// TIA Portal V17 export
// export: Created 2025-03-07T09:19:28.6491986Z, ExportSetting WithDefaults, DisplayName Totally Integrated Automation Portal, DisplayVersion V17 Update 8, DisplayName TIA Portal Openness, DisplayVersion V17 Update 8, DisplayName TIA Portal Version Control Interface, DisplayVersion V17, DisplayName SINAMICS Startdrive Advanced, DisplayVersion V17 SP2, DisplayName SINAMICS Startdrive G110M, G120, G120C, G120D, G120P, G115D, DisplayVersion V17 SP2, DisplayName SINAMICS Startdrive G130, G150, S120, S150, SINAMICS MV, S210, DisplayVersion V17 SP2, DisplayName STEP 7 Professional, DisplayVersion V17 Update 8, DisplayName SINUMERIK ONE STEP 7 Toolbox, DisplayVersion V17 Update 12, DisplayName SINUMERIK 840D sl STEP 7 Toolbox, DisplayVersion V17 Update 12, DisplayName STEP 7 Safety, DisplayVersion V17 Update 6, DisplayName WinCC Advanced, DisplayVersion V17 Update 8
TYPE "LBP_typeTMMagazines"
TITLE = Tool management magazines / Almacenes de gestión de herramientas / Magazine zur Werkzeugverwaltung
// User data type to store the magazine data / Tipo de datos de usuario para guardar los datos de almacén / Anwender-Datentyp zum Speichern der Magazindaten
// stored: IsFailsafeCompliant false
   STRUCT
      MaxSpindleNumber : UInt;   // Maximale Spindelanzahl / Maximum spindle number / Número máximo de cabezales
      NumberOfMagazines : UInt;   // Anzahl aller Magazine einschließlich Belade- und Zwischenspeichermagazine / Number of all magazines including loading and buffer magazines / Número total de almacenes, incluidos almacenes de carga e intermedios
      Magazines : Array[1..64] of Struct   // Alle Magazine einschließlich Belade- und Zwischenspeichermagazine / All magazines including loading and buffer magazines / Todos los almacenes, incluidos almacenes de carga e intermedios
         Number : UInt;   // Magazin-Nummer / Magazine number / Número de almacén
         "Type" : UInt;   // Magazintyp / Magazine type / Tipo de almacén
         Places : UInt;   // Anzahl der Plätze im Magazin / Number of locations in magazine / Número de puestos en el almacén
         TMNumber : UInt;   // Werkzeug-Verwaltungsnummer / Tool management number / Número de gestión de herramientas
      END_STRUCT;
   END_STRUCT;
   // // Magazines[2].Number : Magazin-Nummer / Magazine number / Número de almacén
   // // Magazines[3].Number : Magazin-Nummer / Magazine number / Número de almacén
   // // Magazines[4].Number : Magazin-Nummer / Magazine number / Número de almacén
   // // Magazines[5].Number : Magazin-Nummer / Magazine number / Número de almacén
   // // Magazines[6].Number : Magazin-Nummer / Magazine number / Número de almacén
   // // Magazines[7].Number : Magazin-Nummer / Magazine number / Número de almacén
   // // Magazines[8].Number : Magazin-Nummer / Magazine number / Número de almacén
   // // Magazines[9].Number : Magazin-Nummer / Magazine number / Número de almacén
   // // Magazines[10].Number : Magazin-Nummer / Magazine number / Número de almacén
   // // Magazines[11].Number : Magazin-Nummer / Magazine number / Número de almacén
   // // Magazines[12].Number : Magazin-Nummer / Magazine number / Número de almacén
   // // Magazines[13].Number : Magazin-Nummer / Magazine number / Número de almacén
   // // Magazines[14].Number : Magazin-Nummer / Magazine number / Número de almacén
   // // Magazines[15].Number : Magazin-Nummer / Magazine number / Número de almacén
   // // Magazines[16].Number : Magazin-Nummer / Magazine number / Número de almacén
   // // Magazines[17].Number : Magazin-Nummer / Magazine number / Número de almacén
   // // Magazines[18].Number : Magazin-Nummer / Magazine number / Número de almacén
   // // Magazines[19].Number : Magazin-Nummer / Magazine number / Número de almacén
   // // Magazines[20].Number : Magazin-Nummer / Magazine number / Número de almacén
   // // Magazines[21].Number : Magazin-Nummer / Magazine number / Número de almacén
   // // Magazines[22].Number : Magazin-Nummer / Magazine number / Número de almacén
   // // Magazines[23].Number : Magazin-Nummer / Magazine number / Número de almacén
   // // Magazines[24].Number : Magazin-Nummer / Magazine number / Número de almacén
   // // Magazines[25].Number : Magazin-Nummer / Magazine number / Número de almacén
   // // Magazines[26].Number : Magazin-Nummer / Magazine number / Número de almacén
   // // Magazines[27].Number : Magazin-Nummer / Magazine number / Número de almacén
   // // Magazines[28].Number : Magazin-Nummer / Magazine number / Número de almacén
   // // Magazines[29].Number : Magazin-Nummer / Magazine number / Número de almacén
   // // Magazines[30].Number : Magazin-Nummer / Magazine number / Número de almacén
   // // Magazines[31].Number : Magazin-Nummer / Magazine number / Número de almacén
   // // Magazines[32].Number : Magazin-Nummer / Magazine number / Número de almacén
   // // Magazines[33].Number : Magazin-Nummer / Magazine number / Número de almacén
   // // Magazines[34].Number : Magazin-Nummer / Magazine number / Número de almacén
   // // Magazines[35].Number : Magazin-Nummer / Magazine number / Número de almacén
   // // Magazines[36].Number : Magazin-Nummer / Magazine number / Número de almacén
   // // Magazines[37].Number : Magazin-Nummer / Magazine number / Número de almacén
   // // Magazines[38].Number : Magazin-Nummer / Magazine number / Número de almacén
   // // Magazines[39].Number : Magazin-Nummer / Magazine number / Número de almacén
   // // Magazines[40].Number : Magazin-Nummer / Magazine number / Número de almacén
   // // Magazines[41].Number : Magazin-Nummer / Magazine number / Número de almacén
   // // Magazines[42].Number : Magazin-Nummer / Magazine number / Número de almacén
   // // Magazines[43].Number : Magazin-Nummer / Magazine number / Número de almacén
   // // Magazines[44].Number : Magazin-Nummer / Magazine number / Número de almacén
   // // Magazines[45].Number : Magazin-Nummer / Magazine number / Número de almacén
   // // Magazines[46].Number : Magazin-Nummer / Magazine number / Número de almacén
   // // Magazines[47].Number : Magazin-Nummer / Magazine number / Número de almacén
   // // Magazines[48].Number : Magazin-Nummer / Magazine number / Número de almacén
   // // Magazines[49].Number : Magazin-Nummer / Magazine number / Número de almacén
   // // Magazines[50].Number : Magazin-Nummer / Magazine number / Número de almacén
   // // Magazines[51].Number : Magazin-Nummer / Magazine number / Número de almacén
   // // Magazines[52].Number : Magazin-Nummer / Magazine number / Número de almacén
   // // Magazines[53].Number : Magazin-Nummer / Magazine number / Número de almacén
   // // Magazines[54].Number : Magazin-Nummer / Magazine number / Número de almacén
   // // Magazines[55].Number : Magazin-Nummer / Magazine number / Número de almacén
   // // Magazines[56].Number : Magazin-Nummer / Magazine number / Número de almacén
   // // Magazines[57].Number : Magazin-Nummer / Magazine number / Número de almacén
   // // Magazines[58].Number : Magazin-Nummer / Magazine number / Número de almacén
   // // Magazines[59].Number : Magazin-Nummer / Magazine number / Número de almacén
   // // Magazines[60].Number : Magazin-Nummer / Magazine number / Número de almacén
   // // Magazines[61].Number : Magazin-Nummer / Magazine number / Número de almacén
   // // Magazines[62].Number : Magazin-Nummer / Magazine number / Número de almacén
   // // Magazines[63].Number : Magazin-Nummer / Magazine number / Número de almacén
   // // Magazines[64].Number : Magazin-Nummer / Magazine number / Número de almacén
   // // Magazines[2]."Type" : Magazintyp / Magazine type / Tipo de almacén
   // // Magazines[3]."Type" : Magazintyp / Magazine type / Tipo de almacén
   // // Magazines[4]."Type" : Magazintyp / Magazine type / Tipo de almacén
   // // Magazines[5]."Type" : Magazintyp / Magazine type / Tipo de almacén
   // // Magazines[6]."Type" : Magazintyp / Magazine type / Tipo de almacén
   // // Magazines[7]."Type" : Magazintyp / Magazine type / Tipo de almacén
   // // Magazines[8]."Type" : Magazintyp / Magazine type / Tipo de almacén
   // // Magazines[9]."Type" : Magazintyp / Magazine type / Tipo de almacén
   // // Magazines[10]."Type" : Magazintyp / Magazine type / Tipo de almacén
   // // Magazines[11]."Type" : Magazintyp / Magazine type / Tipo de almacén
   // // Magazines[12]."Type" : Magazintyp / Magazine type / Tipo de almacén
   // // Magazines[13]."Type" : Magazintyp / Magazine type / Tipo de almacén
   // // Magazines[14]."Type" : Magazintyp / Magazine type / Tipo de almacén
   // // Magazines[15]."Type" : Magazintyp / Magazine type / Tipo de almacén
   // // Magazines[16]."Type" : Magazintyp / Magazine type / Tipo de almacén
   // // Magazines[17]."Type" : Magazintyp / Magazine type / Tipo de almacén
   // // Magazines[18]."Type" : Magazintyp / Magazine type / Tipo de almacén
   // // Magazines[19]."Type" : Magazintyp / Magazine type / Tipo de almacén
   // // Magazines[20]."Type" : Magazintyp / Magazine type / Tipo de almacén
   // // Magazines[21]."Type" : Magazintyp / Magazine type / Tipo de almacén
   // // Magazines[22]."Type" : Magazintyp / Magazine type / Tipo de almacén
   // // Magazines[23]."Type" : Magazintyp / Magazine type / Tipo de almacén
   // // Magazines[24]."Type" : Magazintyp / Magazine type / Tipo de almacén
   // // Magazines[25]."Type" : Magazintyp / Magazine type / Tipo de almacén
   // // Magazines[26]."Type" : Magazintyp / Magazine type / Tipo de almacén
   // // Magazines[27]."Type" : Magazintyp / Magazine type / Tipo de almacén
   // // Magazines[28]."Type" : Magazintyp / Magazine type / Tipo de almacén
   // // Magazines[29]."Type" : Magazintyp / Magazine type / Tipo de almacén
   // // Magazines[30]."Type" : Magazintyp / Magazine type / Tipo de almacén
   // // Magazines[31]."Type" : Magazintyp / Magazine type / Tipo de almacén
   // // Magazines[32]."Type" : Magazintyp / Magazine type / Tipo de almacén
   // // Magazines[33]."Type" : Magazintyp / Magazine type / Tipo de almacén
   // // Magazines[34]."Type" : Magazintyp / Magazine type / Tipo de almacén
   // // Magazines[35]."Type" : Magazintyp / Magazine type / Tipo de almacén
   // // Magazines[36]."Type" : Magazintyp / Magazine type / Tipo de almacén
   // // Magazines[37]."Type" : Magazintyp / Magazine type / Tipo de almacén
   // // Magazines[38]."Type" : Magazintyp / Magazine type / Tipo de almacén
   // // Magazines[39]."Type" : Magazintyp / Magazine type / Tipo de almacén
   // // Magazines[40]."Type" : Magazintyp / Magazine type / Tipo de almacén
   // // Magazines[41]."Type" : Magazintyp / Magazine type / Tipo de almacén
   // // Magazines[42]."Type" : Magazintyp / Magazine type / Tipo de almacén
   // // Magazines[43]."Type" : Magazintyp / Magazine type / Tipo de almacén
   // // Magazines[44]."Type" : Magazintyp / Magazine type / Tipo de almacén
   // // Magazines[45]."Type" : Magazintyp / Magazine type / Tipo de almacén
   // // Magazines[46]."Type" : Magazintyp / Magazine type / Tipo de almacén
   // // Magazines[47]."Type" : Magazintyp / Magazine type / Tipo de almacén
   // // Magazines[48]."Type" : Magazintyp / Magazine type / Tipo de almacén
   // // Magazines[49]."Type" : Magazintyp / Magazine type / Tipo de almacén
   // // Magazines[50]."Type" : Magazintyp / Magazine type / Tipo de almacén
   // // Magazines[51]."Type" : Magazintyp / Magazine type / Tipo de almacén
   // // Magazines[52]."Type" : Magazintyp / Magazine type / Tipo de almacén
   // // Magazines[53]."Type" : Magazintyp / Magazine type / Tipo de almacén
   // // Magazines[54]."Type" : Magazintyp / Magazine type / Tipo de almacén
   // // Magazines[55]."Type" : Magazintyp / Magazine type / Tipo de almacén
   // // Magazines[56]."Type" : Magazintyp / Magazine type / Tipo de almacén
   // // Magazines[57]."Type" : Magazintyp / Magazine type / Tipo de almacén
   // // Magazines[58]."Type" : Magazintyp / Magazine type / Tipo de almacén
   // // Magazines[59]."Type" : Magazintyp / Magazine type / Tipo de almacén
   // // Magazines[60]."Type" : Magazintyp / Magazine type / Tipo de almacén
   // // Magazines[61]."Type" : Magazintyp / Magazine type / Tipo de almacén
   // // Magazines[62]."Type" : Magazintyp / Magazine type / Tipo de almacén
   // // Magazines[63]."Type" : Magazintyp / Magazine type / Tipo de almacén
   // // Magazines[64]."Type" : Magazintyp / Magazine type / Tipo de almacén
   // // Magazines[2].Places : Anzahl der Plätze im Magazin / Number of locations in magazine / Número de puestos en el almacén
   // // Magazines[3].Places : Anzahl der Plätze im Magazin / Number of locations in magazine / Número de puestos en el almacén
   // // Magazines[4].Places : Anzahl der Plätze im Magazin / Number of locations in magazine / Número de puestos en el almacén
   // // Magazines[5].Places : Anzahl der Plätze im Magazin / Number of locations in magazine / Número de puestos en el almacén
   // // Magazines[6].Places : Anzahl der Plätze im Magazin / Number of locations in magazine / Número de puestos en el almacén
   // // Magazines[7].Places : Anzahl der Plätze im Magazin / Number of locations in magazine / Número de puestos en el almacén
   // // Magazines[8].Places : Anzahl der Plätze im Magazin / Number of locations in magazine / Número de puestos en el almacén
   // // Magazines[9].Places : Anzahl der Plätze im Magazin / Number of locations in magazine / Número de puestos en el almacén
   // // Magazines[10].Places : Anzahl der Plätze im Magazin / Number of locations in magazine / Número de puestos en el almacén
   // // Magazines[11].Places : Anzahl der Plätze im Magazin / Number of locations in magazine / Número de puestos en el almacén
   // // Magazines[12].Places : Anzahl der Plätze im Magazin / Number of locations in magazine / Número de puestos en el almacén
   // // Magazines[13].Places : Anzahl der Plätze im Magazin / Number of locations in magazine / Número de puestos en el almacén
   // // Magazines[14].Places : Anzahl der Plätze im Magazin / Number of locations in magazine / Número de puestos en el almacén
   // // Magazines[15].Places : Anzahl der Plätze im Magazin / Number of locations in magazine / Número de puestos en el almacén
   // // Magazines[16].Places : Anzahl der Plätze im Magazin / Number of locations in magazine / Número de puestos en el almacén
   // // Magazines[17].Places : Anzahl der Plätze im Magazin / Number of locations in magazine / Número de puestos en el almacén
   // // Magazines[18].Places : Anzahl der Plätze im Magazin / Number of locations in magazine / Número de puestos en el almacén
   // // Magazines[19].Places : Anzahl der Plätze im Magazin / Number of locations in magazine / Número de puestos en el almacén
   // // Magazines[20].Places : Anzahl der Plätze im Magazin / Number of locations in magazine / Número de puestos en el almacén
   // // Magazines[21].Places : Anzahl der Plätze im Magazin / Number of locations in magazine / Número de puestos en el almacén
   // // Magazines[22].Places : Anzahl der Plätze im Magazin / Number of locations in magazine / Número de puestos en el almacén
   // // Magazines[23].Places : Anzahl der Plätze im Magazin / Number of locations in magazine / Número de puestos en el almacén
   // // Magazines[24].Places : Anzahl der Plätze im Magazin / Number of locations in magazine / Número de puestos en el almacén
   // // Magazines[25].Places : Anzahl der Plätze im Magazin / Number of locations in magazine / Número de puestos en el almacén
   // // Magazines[26].Places : Anzahl der Plätze im Magazin / Number of locations in magazine / Número de puestos en el almacén
   // // Magazines[27].Places : Anzahl der Plätze im Magazin / Number of locations in magazine / Número de puestos en el almacén
   // // Magazines[28].Places : Anzahl der Plätze im Magazin / Number of locations in magazine / Número de puestos en el almacén
   // // Magazines[29].Places : Anzahl der Plätze im Magazin / Number of locations in magazine / Número de puestos en el almacén
   // // Magazines[30].Places : Anzahl der Plätze im Magazin / Number of locations in magazine / Número de puestos en el almacén
   // // Magazines[31].Places : Anzahl der Plätze im Magazin / Number of locations in magazine / Número de puestos en el almacén
   // // Magazines[32].Places : Anzahl der Plätze im Magazin / Number of locations in magazine / Número de puestos en el almacén
   // // Magazines[33].Places : Anzahl der Plätze im Magazin / Number of locations in magazine / Número de puestos en el almacén
   // // Magazines[34].Places : Anzahl der Plätze im Magazin / Number of locations in magazine / Número de puestos en el almacén
   // // Magazines[35].Places : Anzahl der Plätze im Magazin / Number of locations in magazine / Número de puestos en el almacén
   // // Magazines[36].Places : Anzahl der Plätze im Magazin / Number of locations in magazine / Número de puestos en el almacén
   // // Magazines[37].Places : Anzahl der Plätze im Magazin / Number of locations in magazine / Número de puestos en el almacén
   // // Magazines[38].Places : Anzahl der Plätze im Magazin / Number of locations in magazine / Número de puestos en el almacén
   // // Magazines[39].Places : Anzahl der Plätze im Magazin / Number of locations in magazine / Número de puestos en el almacén
   // // Magazines[40].Places : Anzahl der Plätze im Magazin / Number of locations in magazine / Número de puestos en el almacén
   // // Magazines[41].Places : Anzahl der Plätze im Magazin / Number of locations in magazine / Número de puestos en el almacén
   // // Magazines[42].Places : Anzahl der Plätze im Magazin / Number of locations in magazine / Número de puestos en el almacén
   // // Magazines[43].Places : Anzahl der Plätze im Magazin / Number of locations in magazine / Número de puestos en el almacén
   // // Magazines[44].Places : Anzahl der Plätze im Magazin / Number of locations in magazine / Número de puestos en el almacén
   // // Magazines[45].Places : Anzahl der Plätze im Magazin / Number of locations in magazine / Número de puestos en el almacén
   // // Magazines[46].Places : Anzahl der Plätze im Magazin / Number of locations in magazine / Número de puestos en el almacén
   // // Magazines[47].Places : Anzahl der Plätze im Magazin / Number of locations in magazine / Número de puestos en el almacén
   // // Magazines[48].Places : Anzahl der Plätze im Magazin / Number of locations in magazine / Número de puestos en el almacén
   // // Magazines[49].Places : Anzahl der Plätze im Magazin / Number of locations in magazine / Número de puestos en el almacén
   // // Magazines[50].Places : Anzahl der Plätze im Magazin / Number of locations in magazine / Número de puestos en el almacén
   // // Magazines[51].Places : Anzahl der Plätze im Magazin / Number of locations in magazine / Número de puestos en el almacén
   // // Magazines[52].Places : Anzahl der Plätze im Magazin / Number of locations in magazine / Número de puestos en el almacén
   // // Magazines[53].Places : Anzahl der Plätze im Magazin / Number of locations in magazine / Número de puestos en el almacén
   // // Magazines[54].Places : Anzahl der Plätze im Magazin / Number of locations in magazine / Número de puestos en el almacén
   // // Magazines[55].Places : Anzahl der Plätze im Magazin / Number of locations in magazine / Número de puestos en el almacén
   // // Magazines[56].Places : Anzahl der Plätze im Magazin / Number of locations in magazine / Número de puestos en el almacén
   // // Magazines[57].Places : Anzahl der Plätze im Magazin / Number of locations in magazine / Número de puestos en el almacén
   // // Magazines[58].Places : Anzahl der Plätze im Magazin / Number of locations in magazine / Número de puestos en el almacén
   // // Magazines[59].Places : Anzahl der Plätze im Magazin / Number of locations in magazine / Número de puestos en el almacén
   // // Magazines[60].Places : Anzahl der Plätze im Magazin / Number of locations in magazine / Número de puestos en el almacén
   // // Magazines[61].Places : Anzahl der Plätze im Magazin / Number of locations in magazine / Número de puestos en el almacén
   // // Magazines[62].Places : Anzahl der Plätze im Magazin / Number of locations in magazine / Número de puestos en el almacén
   // // Magazines[63].Places : Anzahl der Plätze im Magazin / Number of locations in magazine / Número de puestos en el almacén
   // // Magazines[64].Places : Anzahl der Plätze im Magazin / Number of locations in magazine / Número de puestos en el almacén
   // // Magazines[2].TMNumber : Werkzeug-Verwaltungsnummer / Tool management number / Número de gestión de herramientas
   // // Magazines[3].TMNumber : Werkzeug-Verwaltungsnummer / Tool management number / Número de gestión de herramientas
   // // Magazines[4].TMNumber : Werkzeug-Verwaltungsnummer / Tool management number / Número de gestión de herramientas
   // // Magazines[5].TMNumber : Werkzeug-Verwaltungsnummer / Tool management number / Número de gestión de herramientas
   // // Magazines[6].TMNumber : Werkzeug-Verwaltungsnummer / Tool management number / Número de gestión de herramientas
   // // Magazines[7].TMNumber : Werkzeug-Verwaltungsnummer / Tool management number / Número de gestión de herramientas
   // // Magazines[8].TMNumber : Werkzeug-Verwaltungsnummer / Tool management number / Número de gestión de herramientas
   // // Magazines[9].TMNumber : Werkzeug-Verwaltungsnummer / Tool management number / Número de gestión de herramientas
   // // Magazines[10].TMNumber : Werkzeug-Verwaltungsnummer / Tool management number / Número de gestión de herramientas
   // // Magazines[11].TMNumber : Werkzeug-Verwaltungsnummer / Tool management number / Número de gestión de herramientas
   // // Magazines[12].TMNumber : Werkzeug-Verwaltungsnummer / Tool management number / Número de gestión de herramientas
   // // Magazines[13].TMNumber : Werkzeug-Verwaltungsnummer / Tool management number / Número de gestión de herramientas
   // // Magazines[14].TMNumber : Werkzeug-Verwaltungsnummer / Tool management number / Número de gestión de herramientas
   // // Magazines[15].TMNumber : Werkzeug-Verwaltungsnummer / Tool management number / Número de gestión de herramientas
   // // Magazines[16].TMNumber : Werkzeug-Verwaltungsnummer / Tool management number / Número de gestión de herramientas
   // // Magazines[17].TMNumber : Werkzeug-Verwaltungsnummer / Tool management number / Número de gestión de herramientas
   // // Magazines[18].TMNumber : Werkzeug-Verwaltungsnummer / Tool management number / Número de gestión de herramientas
   // // Magazines[19].TMNumber : Werkzeug-Verwaltungsnummer / Tool management number / Número de gestión de herramientas
   // // Magazines[20].TMNumber : Werkzeug-Verwaltungsnummer / Tool management number / Número de gestión de herramientas
   // // Magazines[21].TMNumber : Werkzeug-Verwaltungsnummer / Tool management number / Número de gestión de herramientas
   // // Magazines[22].TMNumber : Werkzeug-Verwaltungsnummer / Tool management number / Número de gestión de herramientas
   // // Magazines[23].TMNumber : Werkzeug-Verwaltungsnummer / Tool management number / Número de gestión de herramientas
   // // Magazines[24].TMNumber : Werkzeug-Verwaltungsnummer / Tool management number / Número de gestión de herramientas
   // // Magazines[25].TMNumber : Werkzeug-Verwaltungsnummer / Tool management number / Número de gestión de herramientas
   // // Magazines[26].TMNumber : Werkzeug-Verwaltungsnummer / Tool management number / Número de gestión de herramientas
   // // Magazines[27].TMNumber : Werkzeug-Verwaltungsnummer / Tool management number / Número de gestión de herramientas
   // // Magazines[28].TMNumber : Werkzeug-Verwaltungsnummer / Tool management number / Número de gestión de herramientas
   // // Magazines[29].TMNumber : Werkzeug-Verwaltungsnummer / Tool management number / Número de gestión de herramientas
   // // Magazines[30].TMNumber : Werkzeug-Verwaltungsnummer / Tool management number / Número de gestión de herramientas
   // // Magazines[31].TMNumber : Werkzeug-Verwaltungsnummer / Tool management number / Número de gestión de herramientas
   // // Magazines[32].TMNumber : Werkzeug-Verwaltungsnummer / Tool management number / Número de gestión de herramientas
   // // Magazines[33].TMNumber : Werkzeug-Verwaltungsnummer / Tool management number / Número de gestión de herramientas
   // // Magazines[34].TMNumber : Werkzeug-Verwaltungsnummer / Tool management number / Número de gestión de herramientas
   // // Magazines[35].TMNumber : Werkzeug-Verwaltungsnummer / Tool management number / Número de gestión de herramientas
   // // Magazines[36].TMNumber : Werkzeug-Verwaltungsnummer / Tool management number / Número de gestión de herramientas
   // // Magazines[37].TMNumber : Werkzeug-Verwaltungsnummer / Tool management number / Número de gestión de herramientas
   // // Magazines[38].TMNumber : Werkzeug-Verwaltungsnummer / Tool management number / Número de gestión de herramientas
   // // Magazines[39].TMNumber : Werkzeug-Verwaltungsnummer / Tool management number / Número de gestión de herramientas
   // // Magazines[40].TMNumber : Werkzeug-Verwaltungsnummer / Tool management number / Número de gestión de herramientas
   // // Magazines[41].TMNumber : Werkzeug-Verwaltungsnummer / Tool management number / Número de gestión de herramientas
   // // Magazines[42].TMNumber : Werkzeug-Verwaltungsnummer / Tool management number / Número de gestión de herramientas
   // // Magazines[43].TMNumber : Werkzeug-Verwaltungsnummer / Tool management number / Número de gestión de herramientas
   // // Magazines[44].TMNumber : Werkzeug-Verwaltungsnummer / Tool management number / Número de gestión de herramientas
   // // Magazines[45].TMNumber : Werkzeug-Verwaltungsnummer / Tool management number / Número de gestión de herramientas
   // // Magazines[46].TMNumber : Werkzeug-Verwaltungsnummer / Tool management number / Número de gestión de herramientas
   // // Magazines[47].TMNumber : Werkzeug-Verwaltungsnummer / Tool management number / Número de gestión de herramientas
   // // Magazines[48].TMNumber : Werkzeug-Verwaltungsnummer / Tool management number / Número de gestión de herramientas
   // // Magazines[49].TMNumber : Werkzeug-Verwaltungsnummer / Tool management number / Número de gestión de herramientas
   // // Magazines[50].TMNumber : Werkzeug-Verwaltungsnummer / Tool management number / Número de gestión de herramientas
   // // Magazines[51].TMNumber : Werkzeug-Verwaltungsnummer / Tool management number / Número de gestión de herramientas
   // // Magazines[52].TMNumber : Werkzeug-Verwaltungsnummer / Tool management number / Número de gestión de herramientas
   // // Magazines[53].TMNumber : Werkzeug-Verwaltungsnummer / Tool management number / Número de gestión de herramientas
   // // Magazines[54].TMNumber : Werkzeug-Verwaltungsnummer / Tool management number / Número de gestión de herramientas
   // // Magazines[55].TMNumber : Werkzeug-Verwaltungsnummer / Tool management number / Número de gestión de herramientas
   // // Magazines[56].TMNumber : Werkzeug-Verwaltungsnummer / Tool management number / Número de gestión de herramientas
   // // Magazines[57].TMNumber : Werkzeug-Verwaltungsnummer / Tool management number / Número de gestión de herramientas
   // // Magazines[58].TMNumber : Werkzeug-Verwaltungsnummer / Tool management number / Número de gestión de herramientas
   // // Magazines[59].TMNumber : Werkzeug-Verwaltungsnummer / Tool management number / Número de gestión de herramientas
   // // Magazines[60].TMNumber : Werkzeug-Verwaltungsnummer / Tool management number / Número de gestión de herramientas
   // // Magazines[61].TMNumber : Werkzeug-Verwaltungsnummer / Tool management number / Número de gestión de herramientas
   // // Magazines[62].TMNumber : Werkzeug-Verwaltungsnummer / Tool management number / Número de gestión de herramientas
   // // Magazines[63].TMNumber : Werkzeug-Verwaltungsnummer / Tool management number / Número de gestión de herramientas
   // // Magazines[64].TMNumber : Werkzeug-Verwaltungsnummer / Tool management number / Número de gestión de herramientas
   // // Magazines[1] : Alle Magazine einschließlich Belade- und Zwischenspeichermagazine / All magazines including loading and buffer magazines / Todos los almacenes, incluidos almacenes de carga e intermedios
   // // Magazines[2] : Alle Magazine einschließlich Belade- und Zwischenspeichermagazine / All magazines including loading and buffer magazines / Todos los almacenes, incluidos almacenes de carga e intermedios
   // // Magazines[3] : Alle Magazine einschließlich Belade- und Zwischenspeichermagazine / All magazines including loading and buffer magazines / Todos los almacenes, incluidos almacenes de carga e intermedios
   // // Magazines[4] : Alle Magazine einschließlich Belade- und Zwischenspeichermagazine / All magazines including loading and buffer magazines / Todos los almacenes, incluidos almacenes de carga e intermedios
   // // Magazines[5] : Alle Magazine einschließlich Belade- und Zwischenspeichermagazine / All magazines including loading and buffer magazines / Todos los almacenes, incluidos almacenes de carga e intermedios
   // // Magazines[6] : Alle Magazine einschließlich Belade- und Zwischenspeichermagazine / All magazines including loading and buffer magazines / Todos los almacenes, incluidos almacenes de carga e intermedios
   // // Magazines[7] : Alle Magazine einschließlich Belade- und Zwischenspeichermagazine / All magazines including loading and buffer magazines / Todos los almacenes, incluidos almacenes de carga e intermedios
   // // Magazines[8] : Alle Magazine einschließlich Belade- und Zwischenspeichermagazine / All magazines including loading and buffer magazines / Todos los almacenes, incluidos almacenes de carga e intermedios
   // // Magazines[9] : Alle Magazine einschließlich Belade- und Zwischenspeichermagazine / All magazines including loading and buffer magazines / Todos los almacenes, incluidos almacenes de carga e intermedios
   // // Magazines[10] : Alle Magazine einschließlich Belade- und Zwischenspeichermagazine / All magazines including loading and buffer magazines / Todos los almacenes, incluidos almacenes de carga e intermedios
   // // Magazines[11] : Alle Magazine einschließlich Belade- und Zwischenspeichermagazine / All magazines including loading and buffer magazines / Todos los almacenes, incluidos almacenes de carga e intermedios
   // // Magazines[12] : Alle Magazine einschließlich Belade- und Zwischenspeichermagazine / All magazines including loading and buffer magazines / Todos los almacenes, incluidos almacenes de carga e intermedios
   // // Magazines[13] : Alle Magazine einschließlich Belade- und Zwischenspeichermagazine / All magazines including loading and buffer magazines / Todos los almacenes, incluidos almacenes de carga e intermedios
   // // Magazines[14] : Alle Magazine einschließlich Belade- und Zwischenspeichermagazine / All magazines including loading and buffer magazines / Todos los almacenes, incluidos almacenes de carga e intermedios
   // // Magazines[15] : Alle Magazine einschließlich Belade- und Zwischenspeichermagazine / All magazines including loading and buffer magazines / Todos los almacenes, incluidos almacenes de carga e intermedios
   // // Magazines[16] : Alle Magazine einschließlich Belade- und Zwischenspeichermagazine / All magazines including loading and buffer magazines / Todos los almacenes, incluidos almacenes de carga e intermedios
   // // Magazines[17] : Alle Magazine einschließlich Belade- und Zwischenspeichermagazine / All magazines including loading and buffer magazines / Todos los almacenes, incluidos almacenes de carga e intermedios
   // // Magazines[18] : Alle Magazine einschließlich Belade- und Zwischenspeichermagazine / All magazines including loading and buffer magazines / Todos los almacenes, incluidos almacenes de carga e intermedios
   // // Magazines[19] : Alle Magazine einschließlich Belade- und Zwischenspeichermagazine / All magazines including loading and buffer magazines / Todos los almacenes, incluidos almacenes de carga e intermedios
   // // Magazines[20] : Alle Magazine einschließlich Belade- und Zwischenspeichermagazine / All magazines including loading and buffer magazines / Todos los almacenes, incluidos almacenes de carga e intermedios
   // // Magazines[21] : Alle Magazine einschließlich Belade- und Zwischenspeichermagazine / All magazines including loading and buffer magazines / Todos los almacenes, incluidos almacenes de carga e intermedios
   // // Magazines[22] : Alle Magazine einschließlich Belade- und Zwischenspeichermagazine / All magazines including loading and buffer magazines / Todos los almacenes, incluidos almacenes de carga e intermedios
   // // Magazines[23] : Alle Magazine einschließlich Belade- und Zwischenspeichermagazine / All magazines including loading and buffer magazines / Todos los almacenes, incluidos almacenes de carga e intermedios
   // // Magazines[24] : Alle Magazine einschließlich Belade- und Zwischenspeichermagazine / All magazines including loading and buffer magazines / Todos los almacenes, incluidos almacenes de carga e intermedios
   // // Magazines[25] : Alle Magazine einschließlich Belade- und Zwischenspeichermagazine / All magazines including loading and buffer magazines / Todos los almacenes, incluidos almacenes de carga e intermedios
   // // Magazines[26] : Alle Magazine einschließlich Belade- und Zwischenspeichermagazine / All magazines including loading and buffer magazines / Todos los almacenes, incluidos almacenes de carga e intermedios
   // // Magazines[27] : Alle Magazine einschließlich Belade- und Zwischenspeichermagazine / All magazines including loading and buffer magazines / Todos los almacenes, incluidos almacenes de carga e intermedios
   // // Magazines[28] : Alle Magazine einschließlich Belade- und Zwischenspeichermagazine / All magazines including loading and buffer magazines / Todos los almacenes, incluidos almacenes de carga e intermedios
   // // Magazines[29] : Alle Magazine einschließlich Belade- und Zwischenspeichermagazine / All magazines including loading and buffer magazines / Todos los almacenes, incluidos almacenes de carga e intermedios
   // // Magazines[30] : Alle Magazine einschließlich Belade- und Zwischenspeichermagazine / All magazines including loading and buffer magazines / Todos los almacenes, incluidos almacenes de carga e intermedios
   // // Magazines[31] : Alle Magazine einschließlich Belade- und Zwischenspeichermagazine / All magazines including loading and buffer magazines / Todos los almacenes, incluidos almacenes de carga e intermedios
   // // Magazines[32] : Alle Magazine einschließlich Belade- und Zwischenspeichermagazine / All magazines including loading and buffer magazines / Todos los almacenes, incluidos almacenes de carga e intermedios
   // // Magazines[33] : Alle Magazine einschließlich Belade- und Zwischenspeichermagazine / All magazines including loading and buffer magazines / Todos los almacenes, incluidos almacenes de carga e intermedios
   // // Magazines[34] : Alle Magazine einschließlich Belade- und Zwischenspeichermagazine / All magazines including loading and buffer magazines / Todos los almacenes, incluidos almacenes de carga e intermedios
   // // Magazines[35] : Alle Magazine einschließlich Belade- und Zwischenspeichermagazine / All magazines including loading and buffer magazines / Todos los almacenes, incluidos almacenes de carga e intermedios
   // // Magazines[36] : Alle Magazine einschließlich Belade- und Zwischenspeichermagazine / All magazines including loading and buffer magazines / Todos los almacenes, incluidos almacenes de carga e intermedios
   // // Magazines[37] : Alle Magazine einschließlich Belade- und Zwischenspeichermagazine / All magazines including loading and buffer magazines / Todos los almacenes, incluidos almacenes de carga e intermedios
   // // Magazines[38] : Alle Magazine einschließlich Belade- und Zwischenspeichermagazine / All magazines including loading and buffer magazines / Todos los almacenes, incluidos almacenes de carga e intermedios
   // // Magazines[39] : Alle Magazine einschließlich Belade- und Zwischenspeichermagazine / All magazines including loading and buffer magazines / Todos los almacenes, incluidos almacenes de carga e intermedios
   // // Magazines[40] : Alle Magazine einschließlich Belade- und Zwischenspeichermagazine / All magazines including loading and buffer magazines / Todos los almacenes, incluidos almacenes de carga e intermedios
   // // Magazines[41] : Alle Magazine einschließlich Belade- und Zwischenspeichermagazine / All magazines including loading and buffer magazines / Todos los almacenes, incluidos almacenes de carga e intermedios
   // // Magazines[42] : Alle Magazine einschließlich Belade- und Zwischenspeichermagazine / All magazines including loading and buffer magazines / Todos los almacenes, incluidos almacenes de carga e intermedios
   // // Magazines[43] : Alle Magazine einschließlich Belade- und Zwischenspeichermagazine / All magazines including loading and buffer magazines / Todos los almacenes, incluidos almacenes de carga e intermedios
   // // Magazines[44] : Alle Magazine einschließlich Belade- und Zwischenspeichermagazine / All magazines including loading and buffer magazines / Todos los almacenes, incluidos almacenes de carga e intermedios
   // // Magazines[45] : Alle Magazine einschließlich Belade- und Zwischenspeichermagazine / All magazines including loading and buffer magazines / Todos los almacenes, incluidos almacenes de carga e intermedios
   // // Magazines[46] : Alle Magazine einschließlich Belade- und Zwischenspeichermagazine / All magazines including loading and buffer magazines / Todos los almacenes, incluidos almacenes de carga e intermedios
   // // Magazines[47] : Alle Magazine einschließlich Belade- und Zwischenspeichermagazine / All magazines including loading and buffer magazines / Todos los almacenes, incluidos almacenes de carga e intermedios
   // // Magazines[48] : Alle Magazine einschließlich Belade- und Zwischenspeichermagazine / All magazines including loading and buffer magazines / Todos los almacenes, incluidos almacenes de carga e intermedios
   // // Magazines[49] : Alle Magazine einschließlich Belade- und Zwischenspeichermagazine / All magazines including loading and buffer magazines / Todos los almacenes, incluidos almacenes de carga e intermedios
   // // Magazines[50] : Alle Magazine einschließlich Belade- und Zwischenspeichermagazine / All magazines including loading and buffer magazines / Todos los almacenes, incluidos almacenes de carga e intermedios
   // // Magazines[51] : Alle Magazine einschließlich Belade- und Zwischenspeichermagazine / All magazines including loading and buffer magazines / Todos los almacenes, incluidos almacenes de carga e intermedios
   // // Magazines[52] : Alle Magazine einschließlich Belade- und Zwischenspeichermagazine / All magazines including loading and buffer magazines / Todos los almacenes, incluidos almacenes de carga e intermedios
   // // Magazines[53] : Alle Magazine einschließlich Belade- und Zwischenspeichermagazine / All magazines including loading and buffer magazines / Todos los almacenes, incluidos almacenes de carga e intermedios
   // // Magazines[54] : Alle Magazine einschließlich Belade- und Zwischenspeichermagazine / All magazines including loading and buffer magazines / Todos los almacenes, incluidos almacenes de carga e intermedios
   // // Magazines[55] : Alle Magazine einschließlich Belade- und Zwischenspeichermagazine / All magazines including loading and buffer magazines / Todos los almacenes, incluidos almacenes de carga e intermedios
   // // Magazines[56] : Alle Magazine einschließlich Belade- und Zwischenspeichermagazine / All magazines including loading and buffer magazines / Todos los almacenes, incluidos almacenes de carga e intermedios
   // // Magazines[57] : Alle Magazine einschließlich Belade- und Zwischenspeichermagazine / All magazines including loading and buffer magazines / Todos los almacenes, incluidos almacenes de carga e intermedios
   // // Magazines[58] : Alle Magazine einschließlich Belade- und Zwischenspeichermagazine / All magazines including loading and buffer magazines / Todos los almacenes, incluidos almacenes de carga e intermedios
   // // Magazines[59] : Alle Magazine einschließlich Belade- und Zwischenspeichermagazine / All magazines including loading and buffer magazines / Todos los almacenes, incluidos almacenes de carga e intermedios
   // // Magazines[60] : Alle Magazine einschließlich Belade- und Zwischenspeichermagazine / All magazines including loading and buffer magazines / Todos los almacenes, incluidos almacenes de carga e intermedios
   // // Magazines[61] : Alle Magazine einschließlich Belade- und Zwischenspeichermagazine / All magazines including loading and buffer magazines / Todos los almacenes, incluidos almacenes de carga e intermedios
   // // Magazines[62] : Alle Magazine einschließlich Belade- und Zwischenspeichermagazine / All magazines including loading and buffer magazines / Todos los almacenes, incluidos almacenes de carga e intermedios
   // // Magazines[63] : Alle Magazine einschließlich Belade- und Zwischenspeichermagazine / All magazines including loading and buffer magazines / Todos los almacenes, incluidos almacenes de carga e intermedios
   // // Magazines[64] : Alle Magazine einschließlich Belade- und Zwischenspeichermagazine / All magazines including loading and buffer magazines / Todos los almacenes, incluidos almacenes de carga e intermedios
END_TYPE
